ABB RobotStudio station: test1_20190225-114432.rsstn

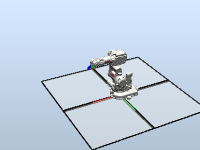
Station test1 (saved by RobotStudio 6.8.8148.134)
Layout (positions relative to the parent item):
  - IRB140_6_81_C_03_2 [mechanism, from Robots\IRB140_6_81_C_G_03.rslib] at (0, 0, 0) mm; joint values [0, 0, 0, 0, 0.5236, 0] (rad or m)
